# EPICS autosave request: BPMApp/Db/TIMRcv_settings.req
$(P)$(R)TimRcvPhaseMeasNavg-SP
$(P)$(R)TimRcvDMTDADeglitch-SP
$(P)$(R)TimRcvDMTDBDeglitch-SP
